INTERFACE ITFBASE EXTENDS I_ITF1

END_INTERFACE

(* stored: Version 1.1.0.1, ProductVersion 3.1.4024.12
   Itf ITFBASE: Id {14fbdfaf-b624-4bbf-a708-c6ee21e1b662} *)
